FUNCTION_BLOCK NOT1 (* Basic Function Block Type *)
  (* Standard: 61499-2 *)
  (* Version 0.0, 9/18/2014, Администратор, nxtControl GmbH, Template *)
  PACKAGE Main;
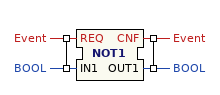
  EVENT_INPUT
    REQ WITH IN1; (* Normal Execution Request *)
  END_EVENT
  EVENT_OUTPUT
    CNF WITH OUT1; (* Execution Confirmation *)
  END_EVENT
  VAR_INPUT
    IN1 : BOOL; (* Input event qualifier *)
  END_VAR
  VAR_OUTPUT
    OUT1 : BOOL; (* Output event qualifier *)
  END_VAR
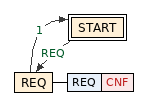
  EC_STATES
    START; (* Initial State *)
    REQ : REQ -> CNF; (* Normal execution *)
  END_STATES
  EC_TRANSITIONS
    START TO REQ := REQ;
    REQ TO START := 1;
  END_TRANSITIONS
  ALGORITHM REQ IN ST:
OUT1 := NOT IN1;
  END_ALGORITHM
END_FUNCTION_BLOCK
